// TIA Portal V19 export
TYPE "LEXCHANGETRAY_typeAxisSimpleControlNodeCommands_2"
// stored: Access Published
   STRUCT
      enableAxis : Bool := FALSE;   // MC_Power: 0: The technology object is disabled / 1: The technology object is enabled / Enable or disable an axis
      resetAxis : Bool := FALSE;   // MC_Reset: Start job with a positive edge / Rising edge: Acknowledgement of technology alarms or reinitialization of the TO
      home : Bool := FALSE;   // MC_Home: Start job with a positive edge / Rising edge: Home an axis
      halt : Bool := FALSE;   // MC_Halt: Start job with a positive edge / Rising edge: Brake an axis until it comes to a standstill
      posAbsolute : Bool := FALSE;   // MC_MoveRelative: Start job with a positive edge / Rising edge: Move an axis to an absolute position
      posRelative : Bool := FALSE;   // MC_MoveAbsolute: Start job with a positive edge / Rising edge: Move an axis relative to its position when execution of the job began
      moveVelocity : Bool := FALSE;   // Rising edge: Move an axis at constant velocity/speed
      jogForward : Bool := FALSE;   // MC_MoveJog: As long as the parameter is TRUE, the axis moves in the positive direction / Rising edge: Move an axis in jog mode (forward); Falling edge: Stop jogging
      jogBackward : Bool := FALSE;   // MC_MoveJog: As long as the parameter is TRUE, the axis moves in the negative direction / Rising edge: Move an axis in jog mode (backward); Falling edge: Stop jogging
      stop : Bool := FALSE;   // Rising edge: Stop all movements of an axis and prevent new motion jobs for the TO. The axis brakes to a standstill and remains switched on
      readValues : Bool := FALSE;   // TRUE: Read values from TO while command is active
      enableTorque : Bool := FALSE;
   END_STRUCT;
END_TYPE
